// TIA Portal V17 export
// export: Created 2025-06-25T13:13:28.9698914Z, ExportSetting WithDefaults, DisplayName Totally Integrated Automation Portal, DisplayVersion V17 Update 8, DisplayName TIA Portal Openness, DisplayVersion V17 Update 8, DisplayName TIA Portal Version Control Interface, DisplayVersion V17, DisplayName STEP 7 Professional, DisplayVersion V17 Update 8, DisplayName STEP 7 Safety, DisplayVersion V17 Update 6, DisplayName WinCC Advanced, DisplayVersion V17 Update 8
TYPE "stSM522_32DQ_Q"
// stored: IsFailsafeCompliant false
   STRUCT
      DQ00 : Bool;
      DQ01 : Bool;
      DQ02 : Bool;
      DQ03 : Bool;
      DQ04 : Bool;
      DQ05 : Bool;
      DQ06 : Bool;
      DQ07 : Bool;
      DQ08 : Bool;
      DQ09 : Bool;
      DQ10 : Bool;
      DQ11 : Bool;
      DQ12 : Bool;
      DQ13 : Bool;
      DQ14 : Bool;
      DQ15 : Bool;
      DQ16 : Bool;
      DQ17 : Bool;
      DQ18 : Bool;
      DQ19 : Bool;
      DQ20 : Bool;
      DQ21 : Bool;
      DQ22 : Bool;
      DQ23 : Bool;
      DQ24 : Bool;
      DQ25 : Bool;
      DQ26 : Bool;
      DQ27 : Bool;
      DQ28 : Bool;
      DQ29 : Bool;
      DQ30 : Bool;
      DQ31 : Bool;
   END_STRUCT;
END_TYPE
